// SIMATIC S7-200 project (STEP 7-Micro/WIN), CPU 222 REL 02.01

SYMBOL_TABLE USUARIO1
PARO             I0.0
MARCHA_1         I0.1
MARCHA_2         I0.2
MARCHA_3         I0.3
E1               Q0.0
E2               Q0.1
END_SYMBOL_TABLE

ORGANIZATION_BLOCK PRINCIPAL:OB1
TITLE=COMENTARIOS DEL PROGRAMA
BEGIN
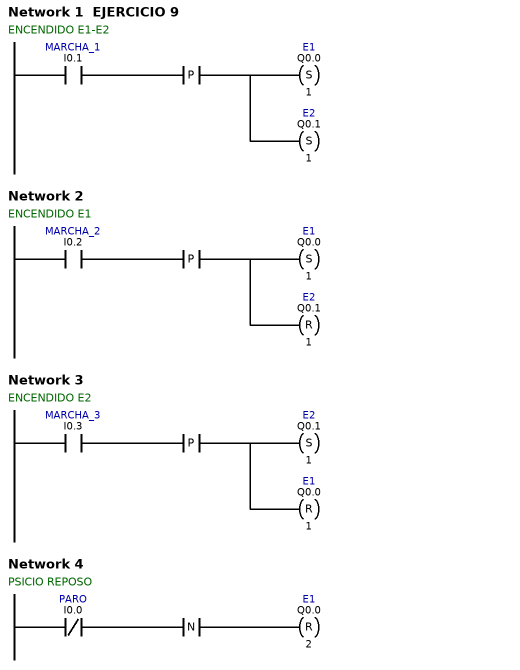
Network 1 // EJERCICIO 9
// ENCENDIDO E1-E2
LD     MARCHA_1:I0.1
EU
S      E1:Q0.0, 1
S      E2:Q0.1, 1
Network 2
// ENCENDIDO E1
// (network saved uncompiled; LAD cells follow)
// row 0: c0 -| |- MARCHA_2:I0.2  c1 -|P|-  v  c2 -(S) E1:Q0.0, 1
// row 1: c1 ^  c2 -(R) E2:Q0.1, 1
Network 3
// ENCENDIDO E2
// (network saved uncompiled; LAD cells follow)
// row 0: c0 -| |- MARCHA_3:I0.3  c1 -|P|-  v  c2 -(S) E2:Q0.1, 1
// row 1: c1 ^  c2 -(R) E1:Q0.0, 1
Network 4
// PSICIO REPOSO
// (network saved uncompiled; LAD cells follow)
// row 0: c0 -|/|- PARO:I0.0  c1 -|N|-  c2 -(R) E1:Q0.0, 2
END_ORGANIZATION_BLOCK
